// TIA Portal V20 export
VAR_GLOBAL   // PLC tag table "Default tag table"
   ResetReactor AT %I0.0 : Bool;
   ServicesOpState AT %I0.1 : Bool;
END_VAR
